// TIA Portal V17 export
// export: Created 2022-03-12T16:05:34.0507696Z, ExportSetting WithDefaults, DisplayName Totally Integrated Automation Portal, DisplayVersion V17, DisplayName TIA Portal Openness, DisplayVersion V17, DisplayName TIA Portal Version Control Interface, DisplayVersion V17, DisplayName STEP 7 Professional, DisplayVersion V17, DisplayName STEP 7 Safety, DisplayVersion V17, DisplayName WinCC Advanced / Unified PC, DisplayVersion V17
TYPE "CPG_typeMessagePrefix"
// stored: IsFailsafeCompliant false
   STRUCT
      messagePrefix : Array[0.."LPMLV30_LANGUAGES_UPPER_LIM"] of String[30];   // Multi-Lingual Message for Prefix (i.e 0=EN, 1=DE, 2=SP/ES, 3=IT, 4=FR)
   END_STRUCT;
END_TYPE
